PROGRAM Auto_Cycle_Fix1
VAR
	Fixture_1 : Fix1_FB;
	TurnTable_0: TurnTable;
	Trunnion_0: Trunnion;
	RollerDoor_0: RollerDoor;
	Robot_Weld_0: Robot_Weld;
	Robot_MH_0: Robot_MH;
END_VAR
VAR // added by the converter: edge detectors and wires of the graphical bodies
    _w1, _w2 : BOOL;
END_VAR

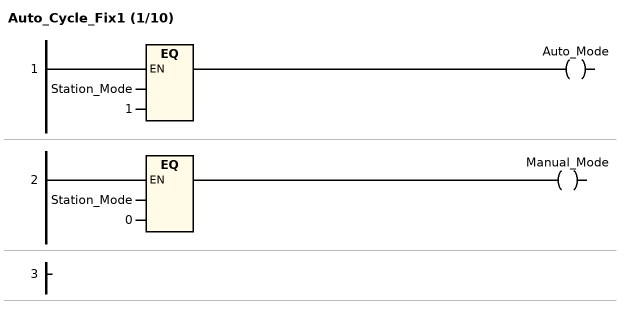
// NETWORK 1
Auto_Mode := Station_Mode = 1;

// NETWORK 2
Manual_Mode := Station_Mode = 0;

// NETWORK 3

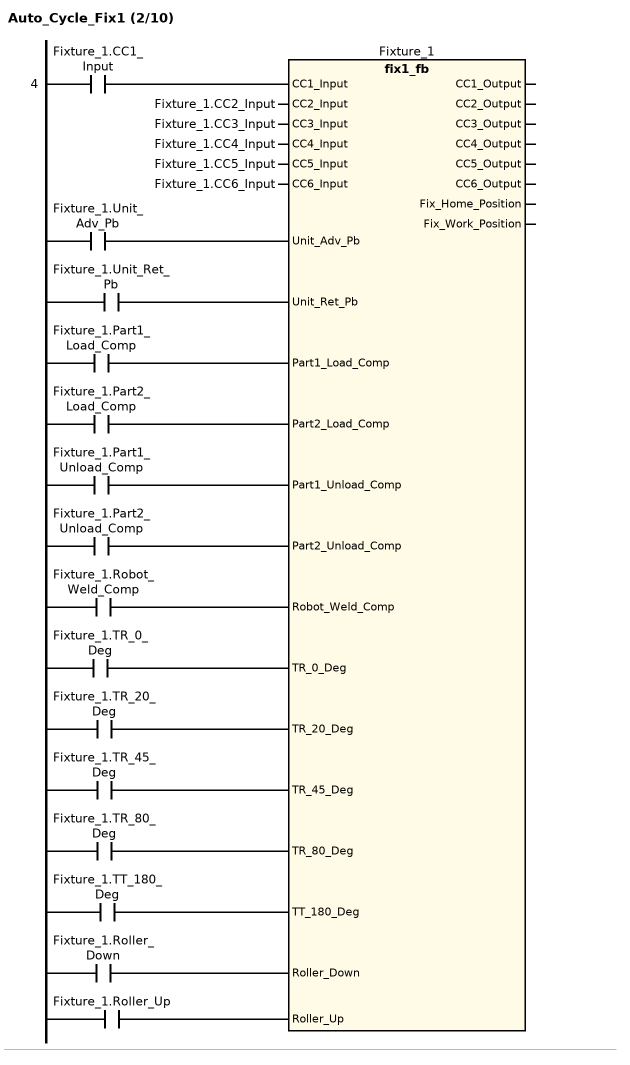
// NETWORK 4
Fixture_1(
    CC1_Input := Fixture_1.CC1_Input,
    CC2_Input := Fixture_1.CC2_Input,
    CC3_Input := Fixture_1.CC3_Input,
    CC4_Input := Fixture_1.CC4_Input,
    CC5_Input := Fixture_1.CC5_Input,
    CC6_Input := Fixture_1.CC6_Input,
    Unit_Adv_Pb := Fixture_1.Unit_Adv_Pb,
    Unit_Ret_Pb := Fixture_1.Unit_Ret_Pb,
    Part1_Load_Comp := Fixture_1.Part1_Load_Comp,
    Part2_Load_Comp := Fixture_1.Part2_Load_Comp,
    Part1_Unload_Comp := Fixture_1.Part1_Unload_Comp,
    Part2_Unload_Comp := Fixture_1.Part2_Unload_Comp,
    Robot_Weld_Comp := Fixture_1.Robot_Weld_Comp,
    TR_0_Deg := Fixture_1.TR_0_Deg,
    TR_20_Deg := Fixture_1.TR_20_Deg,
    TR_45_Deg := Fixture_1.TR_45_Deg,
    TR_80_Deg := Fixture_1.TR_80_Deg,
    TT_180_Deg := Fixture_1.TT_180_Deg,
    Roller_Down := Fixture_1.Roller_Down,
    Roller_Up := Fixture_1.Roller_Up); // fix1_fb

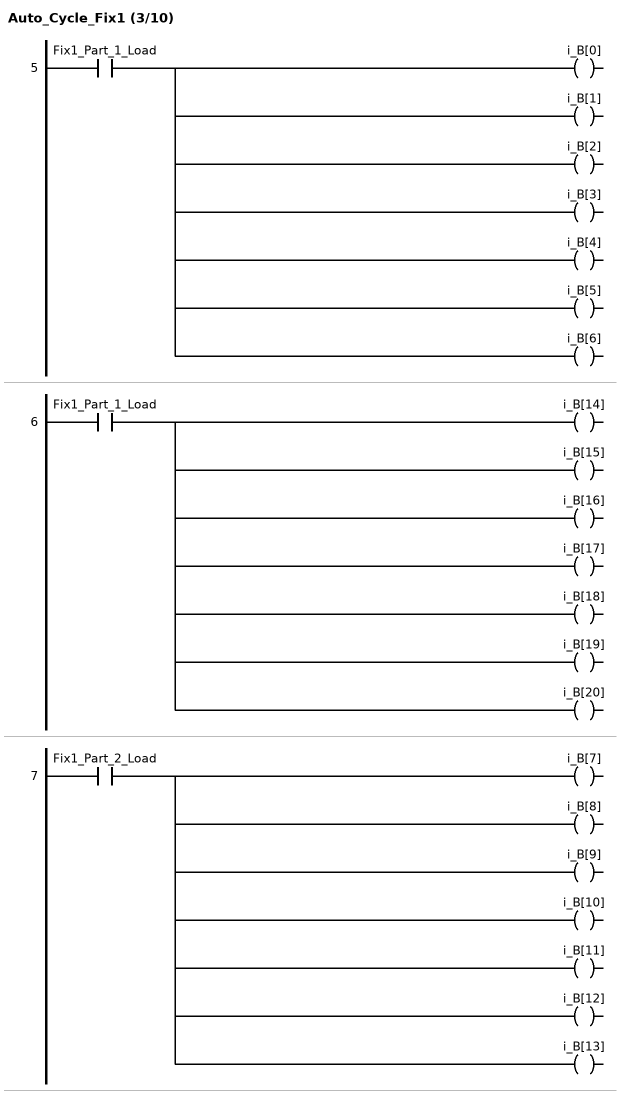
// NETWORK 5
i_B[0] := Fix1_Part_1_Load;
i_B[1] := Fix1_Part_1_Load;
i_B[2] := Fix1_Part_1_Load;
i_B[3] := Fix1_Part_1_Load;
i_B[4] := Fix1_Part_1_Load;
i_B[5] := Fix1_Part_1_Load;
i_B[6] := Fix1_Part_1_Load;

// NETWORK 6
i_B[14] := Fix1_Part_1_Load;
i_B[15] := Fix1_Part_1_Load;
i_B[16] := Fix1_Part_1_Load;
i_B[17] := Fix1_Part_1_Load;
i_B[18] := Fix1_Part_1_Load;
i_B[19] := Fix1_Part_1_Load;
i_B[20] := Fix1_Part_1_Load;

// NETWORK 7
i_B[7] := Fix1_Part_2_Load;
i_B[8] := Fix1_Part_2_Load;
i_B[9] := Fix1_Part_2_Load;
i_B[10] := Fix1_Part_2_Load;
i_B[11] := Fix1_Part_2_Load;
i_B[12] := Fix1_Part_2_Load;
i_B[13] := Fix1_Part_2_Load;

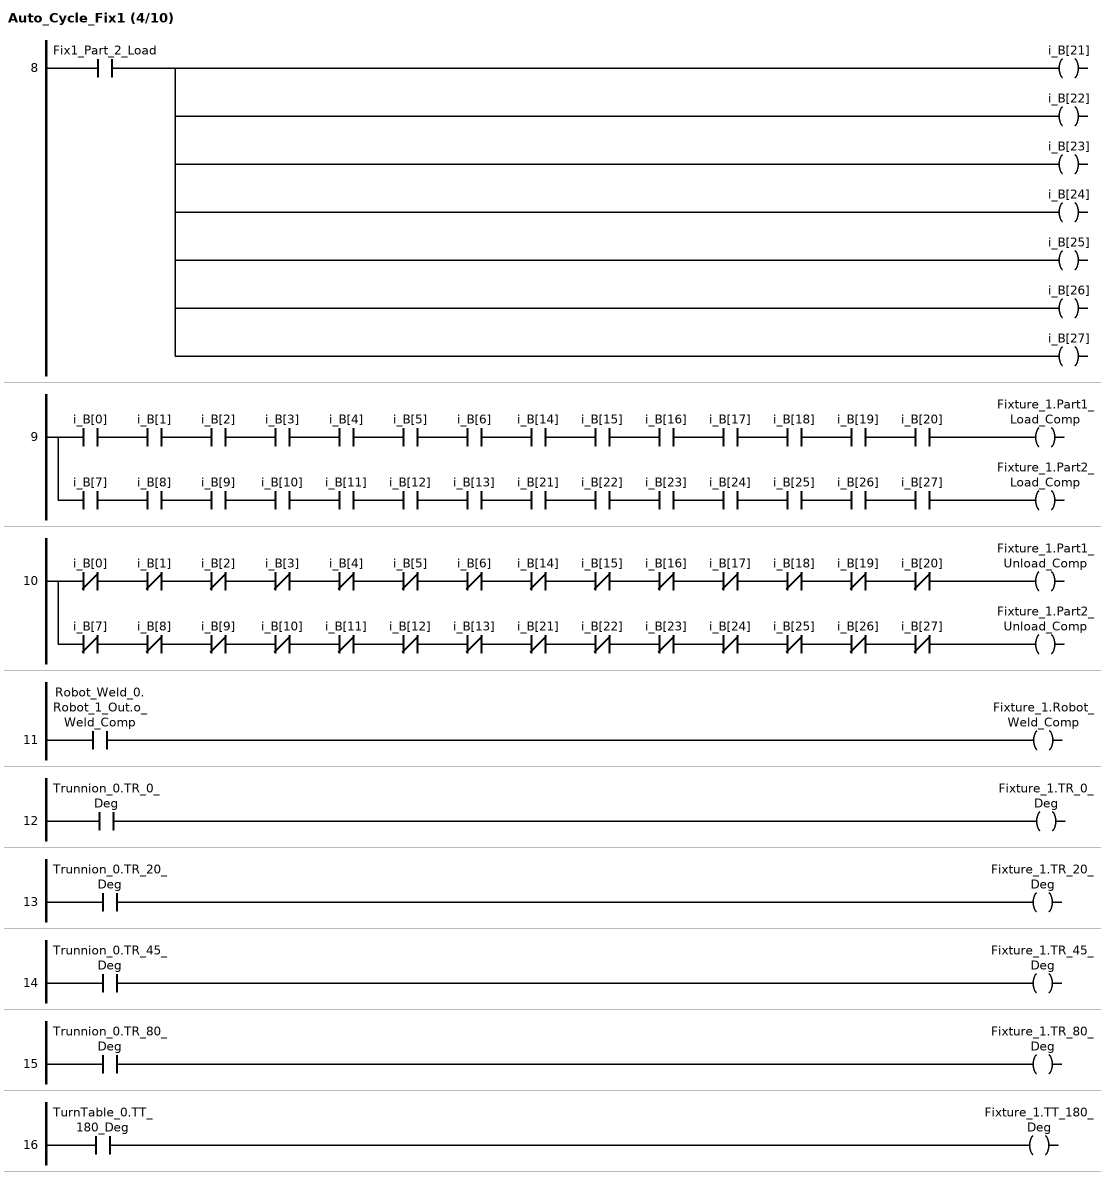
// NETWORK 8
i_B[21] := Fix1_Part_2_Load;
i_B[22] := Fix1_Part_2_Load;
i_B[23] := Fix1_Part_2_Load;
i_B[24] := Fix1_Part_2_Load;
i_B[25] := Fix1_Part_2_Load;
i_B[26] := Fix1_Part_2_Load;
i_B[27] := Fix1_Part_2_Load;

// NETWORK 9
Fixture_1.Part1_Load_Comp := i_B[0] AND i_B[1] AND i_B[2] AND i_B[3] AND i_B[4] AND i_B[5] AND i_B[6] AND i_B[14] AND i_B[15] AND i_B[16] AND i_B[17] AND i_B[18] AND i_B[19] AND i_B[20];
Fixture_1.Part2_Load_Comp := i_B[7] AND i_B[8] AND i_B[9] AND i_B[10] AND i_B[11] AND i_B[12] AND i_B[13] AND i_B[21] AND i_B[22] AND i_B[23] AND i_B[24] AND i_B[25] AND i_B[26] AND i_B[27];

// NETWORK 10
Fixture_1.Part1_Unload_Comp := NOT i_B[0] AND NOT i_B[1] AND NOT i_B[2] AND NOT i_B[3] AND NOT i_B[4] AND NOT i_B[5] AND NOT i_B[6] AND NOT i_B[14] AND NOT i_B[15] AND NOT i_B[16] AND NOT i_B[17] AND NOT i_B[18] AND NOT i_B[19] AND NOT i_B[20];
Fixture_1.Part2_Unload_Comp := NOT i_B[7] AND NOT i_B[8] AND NOT i_B[9] AND NOT i_B[10] AND NOT i_B[11] AND NOT i_B[12] AND NOT i_B[13] AND NOT i_B[21] AND NOT i_B[22] AND NOT i_B[23] AND NOT i_B[24] AND NOT i_B[25] AND NOT i_B[26] AND NOT i_B[27];

// NETWORK 11
Fixture_1.Robot_Weld_Comp := Robot_Weld_0.Robot_1_Out.o_Weld_Comp;

// NETWORK 12
Fixture_1.TR_0_Deg := Trunnion_0.TR_0_Deg;

// NETWORK 13
Fixture_1.TR_20_Deg := Trunnion_0.TR_20_Deg;

// NETWORK 14
Fixture_1.TR_45_Deg := Trunnion_0.TR_45_Deg;

// NETWORK 15
Fixture_1.TR_80_Deg := Trunnion_0.TR_80_Deg;

// NETWORK 16
Fixture_1.TT_180_Deg := TurnTable_0.TT_180_Deg;

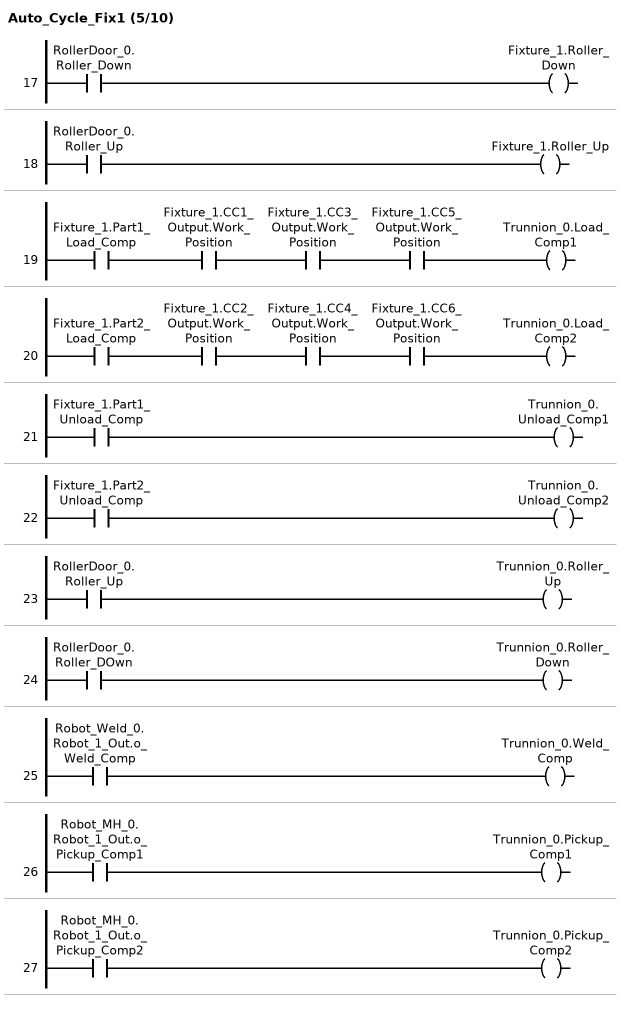
// NETWORK 17
Fixture_1.Roller_Down := RollerDoor_0.Roller_Down;

// NETWORK 18
Fixture_1.Roller_Up := RollerDoor_0.Roller_Up;

// NETWORK 19
Trunnion_0.Load_Comp1 := Fixture_1.Part1_Load_Comp AND Fixture_1.CC1_Output.Work_Position AND Fixture_1.CC3_Output.Work_Position AND Fixture_1.CC5_Output.Work_Position;

// NETWORK 20
Trunnion_0.Load_Comp2 := Fixture_1.Part2_Load_Comp AND Fixture_1.CC2_Output.Work_Position AND Fixture_1.CC4_Output.Work_Position AND Fixture_1.CC6_Output.Work_Position;

// NETWORK 21
Trunnion_0.Unload_Comp1 := Fixture_1.Part1_Unload_Comp;

// NETWORK 22
Trunnion_0.Unload_Comp2 := Fixture_1.Part2_Unload_Comp;

// NETWORK 23
Trunnion_0.Roller_Up := RollerDoor_0.Roller_Up;

// NETWORK 24
Trunnion_0.Roller_Down := RollerDoor_0.Roller_DOwn;

// NETWORK 25
Trunnion_0.Weld_Comp := Robot_Weld_0.Robot_1_Out.o_Weld_Comp;

// NETWORK 26
Trunnion_0.Pickup_Comp1 := Robot_MH_0.Robot_1_Out.o_Pickup_Comp1;

// NETWORK 27
Trunnion_0.Pickup_Comp2 := Robot_MH_0.Robot_1_Out.o_Pickup_Comp2;

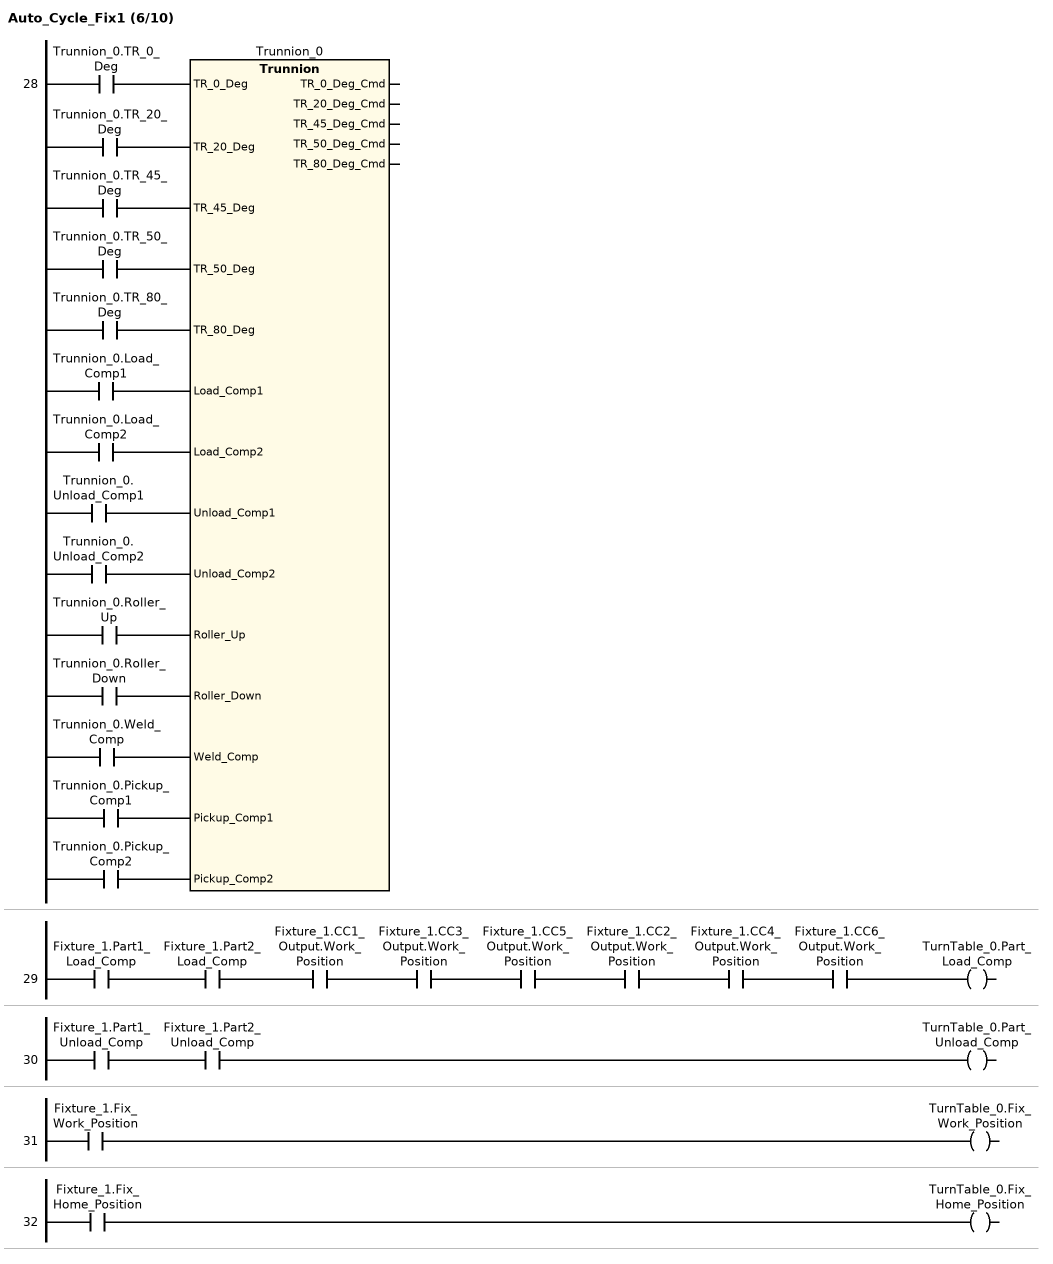
// NETWORK 28
Trunnion_0(
    TR_0_Deg := Trunnion_0.TR_0_Deg,
    TR_20_Deg := Trunnion_0.TR_20_Deg,
    TR_45_Deg := Trunnion_0.TR_45_Deg,
    TR_50_Deg := Trunnion_0.TR_50_Deg,
    TR_80_Deg := Trunnion_0.TR_80_Deg,
    Load_Comp1 := Trunnion_0.Load_Comp1,
    Load_Comp2 := Trunnion_0.Load_Comp2,
    Unload_Comp1 := Trunnion_0.Unload_Comp1,
    Unload_Comp2 := Trunnion_0.Unload_Comp2,
    Roller_Up := Trunnion_0.Roller_Up,
    Roller_Down := Trunnion_0.Roller_Down,
    Weld_Comp := Trunnion_0.Weld_Comp,
    Pickup_Comp1 := Trunnion_0.Pickup_Comp1,
    Pickup_Comp2 := Trunnion_0.Pickup_Comp2); // Trunnion

// NETWORK 29
TurnTable_0.Part_Load_Comp := Fixture_1.Part1_Load_Comp AND Fixture_1.Part2_Load_Comp AND Fixture_1.CC1_Output.Work_Position AND Fixture_1.CC3_Output.Work_Position AND Fixture_1.CC5_Output.Work_Position AND Fixture_1.CC2_Output.Work_Position AND Fixture_1.CC4_Output.Work_Position AND Fixture_1.CC6_Output.Work_Position;

// NETWORK 30
TurnTable_0.Part_Unload_Comp := Fixture_1.Part1_Unload_Comp AND Fixture_1.Part2_Unload_Comp;

// NETWORK 31
TurnTable_0.Fix_Work_Position := Fixture_1.Fix_Work_Position;

// NETWORK 32
TurnTable_0.Fix_Home_Position := Fixture_1.Fix_Home_Position;

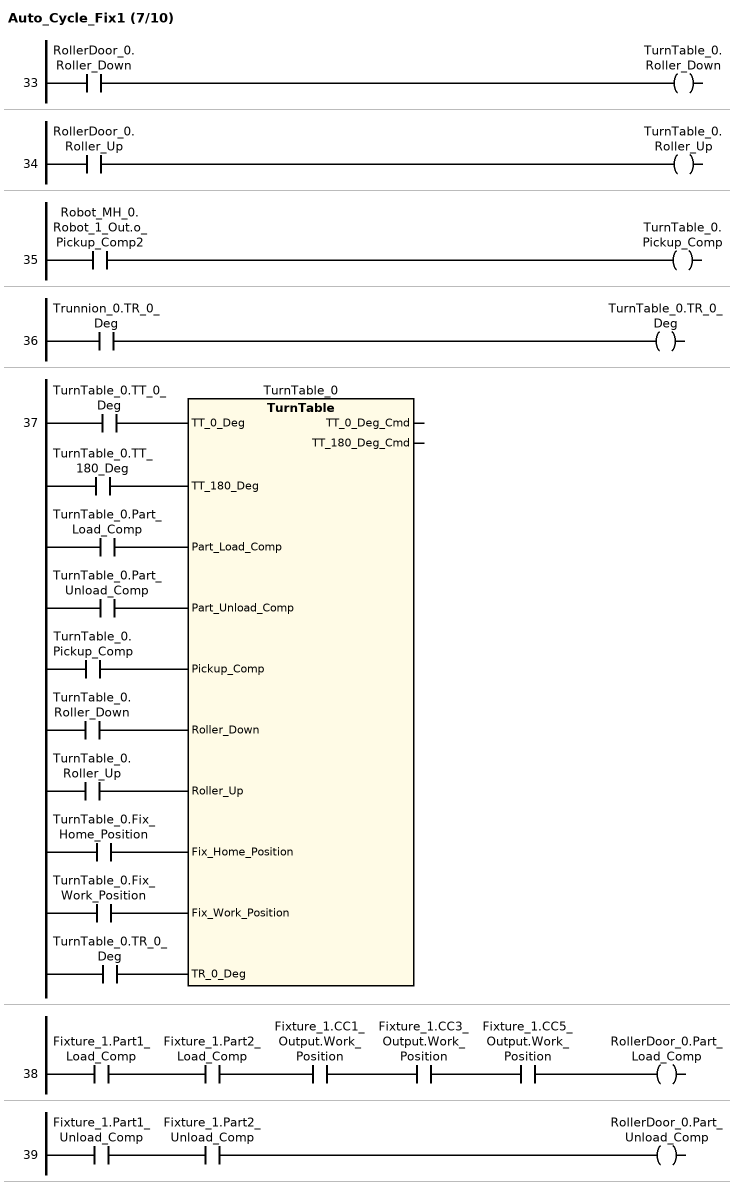
// NETWORK 33
TurnTable_0.Roller_Down := RollerDoor_0.Roller_Down;

// NETWORK 34
TurnTable_0.Roller_Up := RollerDoor_0.Roller_Up;

// NETWORK 35
TurnTable_0.Pickup_Comp := Robot_MH_0.Robot_1_Out.o_Pickup_Comp2;

// NETWORK 36
TurnTable_0.TR_0_Deg := Trunnion_0.TR_0_Deg;

// NETWORK 37
TurnTable_0(
    TT_0_Deg := TurnTable_0.TT_0_Deg,
    TT_180_Deg := TurnTable_0.TT_180_Deg,
    Part_Load_Comp := TurnTable_0.Part_Load_Comp,
    Part_Unload_Comp := TurnTable_0.Part_Unload_Comp,
    Pickup_Comp := TurnTable_0.Pickup_Comp,
    Roller_Down := TurnTable_0.Roller_Down,
    Roller_Up := TurnTable_0.Roller_Up,
    Fix_Home_Position := TurnTable_0.Fix_Home_Position,
    Fix_Work_Position := TurnTable_0.Fix_Work_Position,
    TR_0_Deg := TurnTable_0.TR_0_Deg); // TurnTable

// NETWORK 38
RollerDoor_0.Part_Load_Comp := Fixture_1.Part1_Load_Comp AND Fixture_1.Part2_Load_Comp AND Fixture_1.CC1_Output.Work_Position AND Fixture_1.CC3_Output.Work_Position AND Fixture_1.CC5_Output.Work_Position;

// NETWORK 39
RollerDoor_0.Part_Unload_Comp := Fixture_1.Part1_Unload_Comp AND Fixture_1.Part2_Unload_Comp;

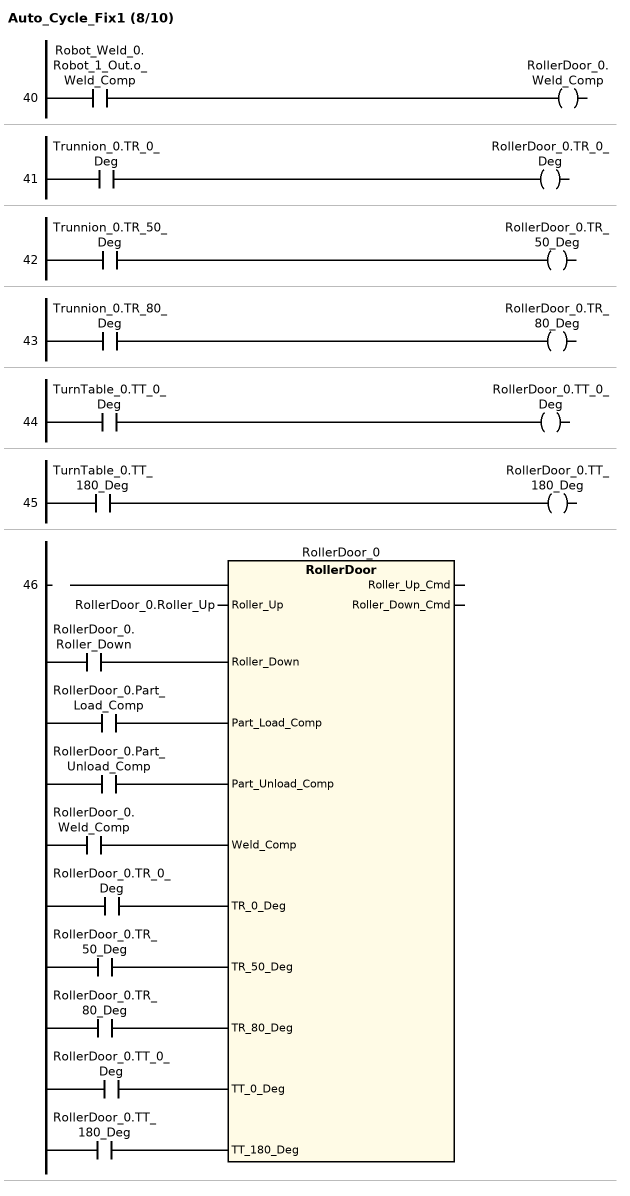
// NETWORK 40
RollerDoor_0.Weld_Comp := Robot_Weld_0.Robot_1_Out.o_Weld_Comp;

// NETWORK 41
RollerDoor_0.TR_0_Deg := Trunnion_0.TR_0_Deg;

// NETWORK 42
RollerDoor_0.TR_50_Deg := Trunnion_0.TR_50_Deg;

// NETWORK 43
RollerDoor_0.TR_80_Deg := Trunnion_0.TR_80_Deg;

// NETWORK 44
RollerDoor_0.TT_0_Deg := TurnTable_0.TT_0_Deg;

// NETWORK 45
RollerDoor_0.TT_180_Deg := TurnTable_0.TT_180_Deg;

// NETWORK 46
RollerDoor_0(
    Roller_Up := RollerDoor_0.Roller_Up,
    Roller_Down := RollerDoor_0.Roller_Down,
    Part_Load_Comp := RollerDoor_0.Part_Load_Comp,
    Part_Unload_Comp := RollerDoor_0.Part_Unload_Comp,
    Weld_Comp := RollerDoor_0.Weld_Comp,
    TR_0_Deg := RollerDoor_0.TR_0_Deg,
    TR_50_Deg := RollerDoor_0.TR_50_Deg,
    TR_80_Deg := RollerDoor_0.TR_80_Deg,
    TT_0_Deg := RollerDoor_0.TT_0_Deg,
    TT_180_Deg := RollerDoor_0.TT_180_Deg); // RollerDoor

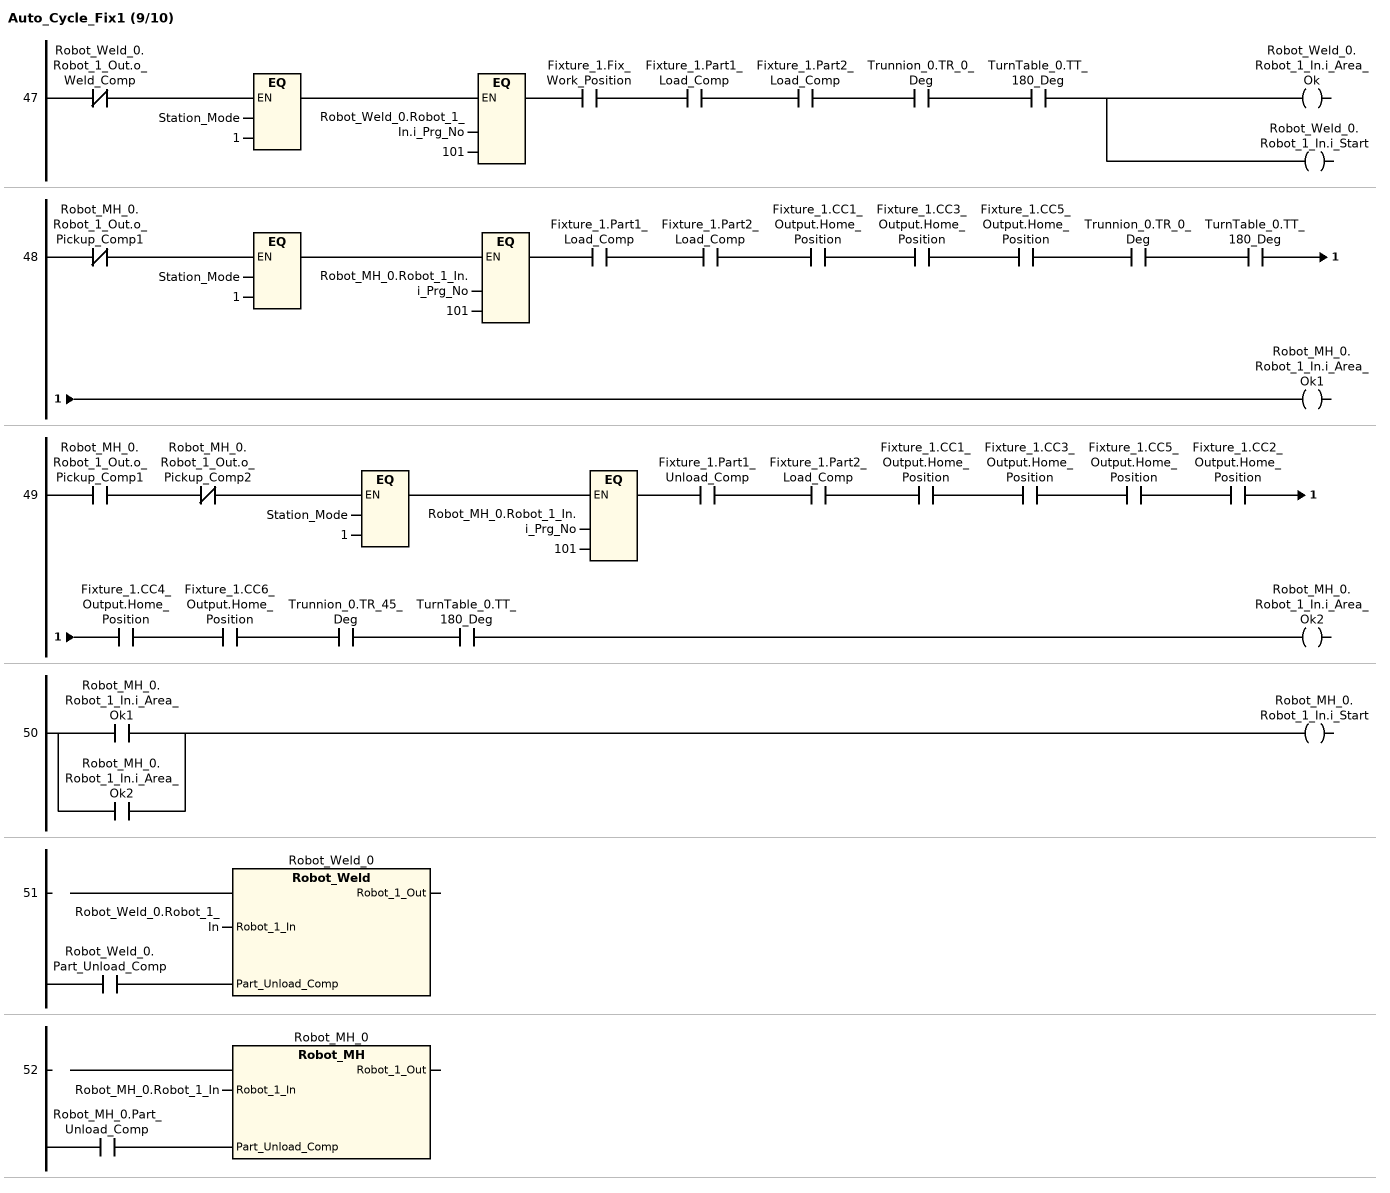
// NETWORK 47
_w1 := (NOT Robot_Weld_0.Robot_1_Out.o_Weld_Comp AND Station_Mode = 1 AND Robot_Weld_0.Robot_1_In.i_Prg_No = 101) AND Fixture_1.Fix_Work_Position AND Fixture_1.Part1_Load_Comp AND Fixture_1.Part2_Load_Comp AND Trunnion_0.TR_0_Deg AND TurnTable_0.TT_180_Deg;
Robot_Weld_0.Robot_1_In.i_Area_Ok := _w1;
Robot_Weld_0.Robot_1_In.i_Start := _w1;

// NETWORK 48
Robot_MH_0.Robot_1_In.i_Area_Ok1 := (NOT Robot_MH_0.Robot_1_Out.o_Pickup_Comp1 AND Station_Mode = 1 AND Robot_MH_0.Robot_1_In.i_Prg_No = 101) AND Fixture_1.Part1_Load_Comp AND Fixture_1.Part2_Load_Comp AND Fixture_1.CC1_Output.Home_Position AND Fixture_1.CC3_Output.Home_Position AND Fixture_1.CC5_Output.Home_Position AND Trunnion_0.TR_0_Deg AND TurnTable_0.TT_180_Deg;

// NETWORK 49
Robot_MH_0.Robot_1_In.i_Area_Ok2 := (Robot_MH_0.Robot_1_Out.o_Pickup_Comp1 AND NOT Robot_MH_0.Robot_1_Out.o_Pickup_Comp2 AND Station_Mode = 1 AND Robot_MH_0.Robot_1_In.i_Prg_No = 101) AND Fixture_1.Part1_Unload_Comp AND Fixture_1.Part2_Load_Comp AND Fixture_1.CC1_Output.Home_Position AND Fixture_1.CC3_Output.Home_Position AND Fixture_1.CC5_Output.Home_Position AND Fixture_1.CC2_Output.Home_Position AND Fixture_1.CC4_Output.Home_Position AND Fixture_1.CC6_Output.Home_Position AND Trunnion_0.TR_45_Deg AND TurnTable_0.TT_180_Deg;

// NETWORK 50
Robot_MH_0.Robot_1_In.i_Start := Robot_MH_0.Robot_1_In.i_Area_Ok1 OR Robot_MH_0.Robot_1_In.i_Area_Ok2;

// NETWORK 51
Robot_Weld_0(Robot_1_In := Robot_Weld_0.Robot_1_In, Part_Unload_Comp := Robot_Weld_0.Part_Unload_Comp); // Robot_Weld

// NETWORK 52
Robot_MH_0(Robot_1_In := Robot_MH_0.Robot_1_In, Part_Unload_Comp := Robot_MH_0.Part_Unload_Comp); // Robot_MH

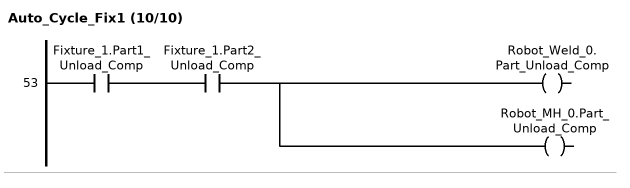
// NETWORK 53
_w2 := Fixture_1.Part1_Unload_Comp AND Fixture_1.Part2_Unload_Comp;
Robot_Weld_0.Part_Unload_Comp := _w2;
Robot_MH_0.Part_Unload_Comp := _w2;

END_PROGRAM

(* stored: Version 1.1.0.1, ProductVersion 3.1.4024.16
   POU Auto_Cycle_Fix1: Id {3cfd5fcc-4e92-4dbb-a127-d131b41b4be0}, SpecialFunc None *)
